Fanuc TP program (LS listing): CORR_NABI828_NIEO.LS

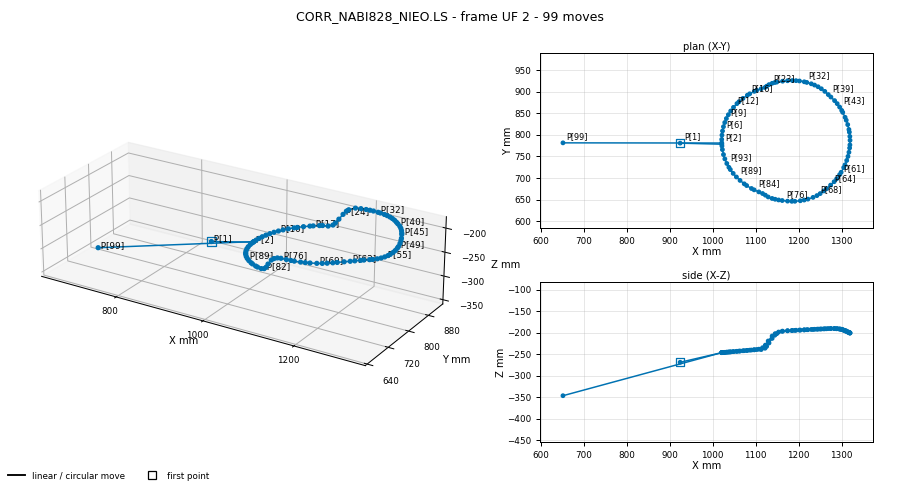
[picture p0: tool path of CORR_NABI828_NIEO.LS in frame UF 2, 99 of 99 moves have a stored position in this frame; points joined in program order, loops and branches not executed]
/PROG  CORR_NABI828_NIEO
/ATTR
OWNER		= MNEDITOR;
COMMENT		= "WeldPRO Auto-Gen";
PROG_SIZE	= 7125;
CREATE		= DATE 26-07-31  TIME 09:44:06;
MODIFIED	= DATE 26-07-31  TIME 10:09:20;
FILE_NAME	= CORR_NAB;
VERSION		= 0;
LINE_COUNT	= 113;
MEMORY_SIZE	= 7445;
PROTECT		= READ_WRITE;
TCD:  STACK_SIZE	= 0,
      TASK_PRIORITY	= 50,
      TIME_SLICE	= 0,
      BUSY_LAMP_OFF	= 0,
      ABORT_REQUEST	= 0,
      PAUSE_REQUEST	= 0;
DEFAULT_GROUP	= 1,*,*,*,*;
CONTROL_CODE	= 00000000 00000000;
/APPL
/MN
   1:  !WeldPRO Auto-Generated TPP ;
   2:  !TOR_XL_2026, TOR_xl_2907 ;
   3:   ;
   4:  UFRAME_NUM=2 ;
   5:  UTOOL_NUM=2 ;
   6:  !Feature Approach ;
   7:J P[1] 100% FINE    ;
   8:   ;
   9:  !Segment1 ;
  10:L P[2] 2000mm/sec FINE    ;
  11:   ;
  12:  CALL LASER_OFF    ;
  13:L P[3] R[23:moving]mm/sec CNT100    ;
  14:L P[4] R[23:moving]mm/sec CNT100    ;
  15:L P[5] R[23:moving]mm/sec CNT100    ;
  16:L P[6] R[23:moving]mm/sec CNT100    ;
  17:L P[7] R[23:moving]mm/sec CNT100    ;
  18:L P[8] R[23:moving]mm/sec CNT100    ;
  19:L P[9] R[23:moving]mm/sec CNT100    ;
  20:L P[10] R[23:moving]mm/sec CNT100    ;
  21:L P[11] R[23:moving]mm/sec CNT100    ;
  22:L P[12] R[23:moving]mm/sec CNT100    ;
  23:L P[13] R[23:moving]mm/sec CNT100    ;
  24:L P[14] R[23:moving]mm/sec CNT100    ;
  25:L P[15] R[23:moving]mm/sec CNT100    ;
  26:L P[16] R[23:moving]mm/sec CNT100    ;
  27:L P[17] R[23:moving]mm/sec CNT100    ;
  28:L P[18] R[23:moving]mm/sec CNT100    ;
  29:L P[19] R[23:moving]mm/sec CNT100    ;
  30:L P[20] R[23:moving]mm/sec CNT100    ;
  31:L P[21] R[23:moving]mm/sec CNT100    ;
  32:L P[22] R[23:moving]mm/sec CNT100    ;
  33:L P[23] R[23:moving]mm/sec CNT100    ;
  34:L P[24] R[23:moving]mm/sec CNT100    ;
  35:L P[25] R[23:moving]mm/sec CNT100    ;
  36:L P[26] R[23:moving]mm/sec CNT100    ;
  37:L P[27] R[23:moving]mm/sec CNT100    ;
  38:L P[28] R[23:moving]mm/sec CNT100    ;
  39:L P[29] R[23:moving]mm/sec CNT100    ;
  40:L P[30] R[23:moving]mm/sec CNT100    ;
  41:L P[31] R[23:moving]mm/sec CNT100    ;
  42:L P[32] R[23:moving]mm/sec CNT100    ;
  43:L P[33] R[23:moving]mm/sec CNT100    ;
  44:L P[34] R[23:moving]mm/sec CNT100    ;
  45:L P[35] R[23:moving]mm/sec CNT100    ;
  46:L P[36] R[23:moving]mm/sec CNT100    ;
  47:L P[37] R[23:moving]mm/sec CNT100    ;
  48:L P[38] R[23:moving]mm/sec CNT100    ;
  49:L P[39] R[23:moving]mm/sec CNT100    ;
  50:L P[40] R[23:moving]mm/sec CNT100    ;
  51:L P[41] R[23:moving]mm/sec CNT100    ;
  52:L P[42] R[23:moving]mm/sec CNT100    ;
  53:L P[43] R[23:moving]mm/sec CNT100    ;
  54:L P[44] R[23:moving]mm/sec CNT100    ;
  55:L P[45] R[23:moving]mm/sec CNT100    ;
  56:L P[46] R[23:moving]mm/sec CNT100    ;
  57:L P[47] R[23:moving]mm/sec CNT100    ;
  58:L P[48] R[23:moving]mm/sec CNT100    ;
  59:L P[49] R[23:moving]mm/sec CNT100    ;
  60:L P[50] R[23:moving]mm/sec CNT100    ;
  61:L P[51] R[23:moving]mm/sec CNT100    ;
  62:L P[52] R[23:moving]mm/sec CNT100    ;
  63:L P[53] R[23:moving]mm/sec CNT100    ;
  64:L P[54] R[23:moving]mm/sec CNT100    ;
  65:L P[55] R[23:moving]mm/sec CNT100    ;
  66:L P[56] R[23:moving]mm/sec CNT100    ;
  67:L P[57] R[23:moving]mm/sec CNT100    ;
  68:L P[58] R[23:moving]mm/sec CNT100    ;
  69:L P[59] R[23:moving]mm/sec CNT100    ;
  70:L P[60] R[23:moving]mm/sec CNT100    ;
  71:L P[61] R[23:moving]mm/sec CNT100    ;
  72:L P[62] R[23:moving]mm/sec CNT100    ;
  73:L P[63] R[23:moving]mm/sec CNT100    ;
  74:L P[64] R[23:moving]mm/sec CNT100    ;
  75:L P[65] R[23:moving]mm/sec CNT100    ;
  76:L P[66] R[23:moving]mm/sec CNT100    ;
  77:L P[67] R[23:moving]mm/sec CNT100    ;
  78:L P[68] R[23:moving]mm/sec CNT100    ;
  79:L P[69] R[23:moving]mm/sec CNT100    ;
  80:L P[70] R[23:moving]mm/sec CNT100    ;
  81:L P[71] R[23:moving]mm/sec CNT100    ;
  82:L P[72] R[23:moving]mm/sec CNT100    ;
  83:L P[73] R[23:moving]mm/sec CNT100    ;
  84:L P[74] R[23:moving]mm/sec CNT100    ;
  85:L P[75] R[23:moving]mm/sec CNT100    ;
  86:L P[76] R[23:moving]mm/sec CNT100    ;
  87:L P[77] R[23:moving]mm/sec CNT100    ;
  88:L P[78] R[23:moving]mm/sec CNT100    ;
  89:L P[79] R[23:moving]mm/sec CNT100    ;
  90:L P[80] R[23:moving]mm/sec CNT100    ;
  91:L P[81] R[23:moving]mm/sec CNT100    ;
  92:L P[82] R[23:moving]mm/sec CNT100    ;
  93:L P[83] R[23:moving]mm/sec CNT100    ;
  94:L P[84] R[23:moving]mm/sec CNT100    ;
  95:L P[85] R[23:moving]mm/sec CNT100    ;
  96:L P[86] R[23:moving]mm/sec CNT100    ;
  97:L P[87] R[23:moving]mm/sec CNT100    ;
  98:L P[88] R[23:moving]mm/sec CNT100    ;
  99:L P[89] R[23:moving]mm/sec CNT100    ;
 100:L P[90] R[23:moving]mm/sec CNT100    ;
 101:L P[91] R[23:moving]mm/sec CNT100    ;
 102:L P[92] R[23:moving]mm/sec CNT100    ;
 103:L P[93] R[23:moving]mm/sec CNT100    ;
 104:L P[94] R[23:moving]mm/sec CNT100    ;
 105:L P[95] R[23:moving]mm/sec CNT100    ;
 106:L P[96] R[23:moving]mm/sec CNT100    ;
 107:L P[97] R[23:moving]mm/sec CNT100    ;
 108:L P[98] R[23:moving]mm/sec FINE    ;
 109:  CALL LASER_OFF    ;
 110:   ;
 111:  !Feature Retreat ;
 112:L P[99] 2000mm/sec FINE    ;
 113:  CALL ROTATE    ;
/POS
P[1]{
   GP1:
	UF : 2, UT : 2,		CONFIG : 'F D T, 0, 0, 0',
	X =   924.335  mm,	Y =   780.986  mm,	Z =  -268.284  mm,
	W =  -106.495 deg,	P =   -15.000 deg,	R =    94.234 deg
};
P[2]{
   GP1:
	UF : 2, UT : 2,		CONFIG : 'F D T, 0, 0, 0',
	X =  1021.169  mm,	Y =   778.543  mm,	Z =  -245.849  mm,
	W =  -106.497 deg,	P =   -14.995 deg,	R =    94.216 deg
};
P[3]{
   GP1:
	UF : 2, UT : 2,		CONFIG : 'F D T, 0, 0, 0',
	X =  1021.011  mm,	Y =   781.278  mm,	Z =  -245.859  mm,
	W =  -106.499 deg,	P =   -14.997 deg,	R =    94.226 deg
};
P[4]{
   GP1:
	UF : 2, UT : 2,		CONFIG : 'F D T, 0, 0, 0',
	X =  1020.925  mm,	Y =   789.680  mm,	Z =  -245.860  mm,
	W =  -106.492 deg,	P =   -15.098 deg,	R =    90.372 deg
};
P[5]{
   GP1:
	UF : 2, UT : 2,		CONFIG : 'F D T, 0, 0, 0',
	X =  1021.526  mm,	Y =   799.646  mm,	Z =  -245.805  mm,
	W =  -106.481 deg,	P =   -15.218 deg,	R =    85.605 deg
};
P[6]{
   GP1:
	UF : 2, UT : 2,		CONFIG : 'F D T, 0, 0, 0',
	X =  1022.834  mm,	Y =   809.284  mm,	Z =  -245.689  mm,
	W =  -106.456 deg,	P =   -15.335 deg,	R =    80.815 deg
};
P[7]{
   GP1:
	UF : 2, UT : 2,		CONFIG : 'F D T, 0, 0, 0',
	X =  1025.009  mm,	Y =   819.272  mm,	Z =  -245.496  mm,
	W =  -106.423 deg,	P =   -15.450 deg,	R =    76.090 deg
};
P[8]{
   GP1:
	UF : 2, UT : 2,		CONFIG : 'F D T, 0, 0, 0',
	X =  1027.996  mm,	Y =   828.917  mm,	Z =  -245.233  mm,
	W =  -106.378 deg,	P =   -15.565 deg,	R =    71.217 deg
};
P[9]{
   GP1:
	UF : 2, UT : 2,		CONFIG : 'F D T, 0, 0, 0',
	X =  1031.797  mm,	Y =   838.208  mm,	Z =  -244.899  mm,
	W =  -106.322 deg,	P =   -15.679 deg,	R =    66.207 deg
};
P[10]{
   GP1:
	UF : 2, UT : 2,		CONFIG : 'F D T, 0, 0, 0',
	X =  1036.420  mm,	Y =   847.146  mm,	Z =  -244.496  mm,
	W =  -106.254 deg,	P =   -15.791 deg,	R =    61.015 deg
};
P[11]{
   GP1:
	UF : 2, UT : 2,		CONFIG : 'F D T, 0, 0, 0',
	X =  1041.832  mm,	Y =   855.675  mm,	Z =  -244.021  mm,
	W =  -106.177 deg,	P =   -15.894 deg,	R =    55.979 deg
};
P[12]{
   GP1:
	UF : 2, UT : 2,		CONFIG : 'F D T, 0, 0, 0',
	X =  1048.352  mm,	Y =   864.193  mm,	Z =  -243.446  mm,
	W =  -106.096 deg,	P =   -15.986 deg,	R =    51.162 deg
};
P[13]{
   GP1:
	UF : 2, UT : 2,		CONFIG : 'F D T, 0, 0, 0',
	X =  1056.339  mm,	Y =   872.875  mm,	Z =  -242.736  mm,
	W =  -106.012 deg,	P =   -16.066 deg,	R =    46.632 deg
};
P[14]{
   GP1:
	UF : 2, UT : 2,		CONFIG : 'F D T, 0, 0, 0',
	X =  1061.049  mm,	Y =   877.307  mm,	Z =  -242.336  mm,
	W =  -105.919 deg,	P =   -16.142 deg,	R =    41.952 deg
};
P[15]{
   GP1:
	UF : 2, UT : 2,		CONFIG : 'F D T, 0, 0, 0',
	X =  1070.354  mm,	Y =   885.100  mm,	Z =  -241.489  mm,
	W =  -105.870 deg,	P =   -16.177 deg,	R =    39.609 deg
};
P[16]{
   GP1:
	UF : 2, UT : 2,		CONFIG : 'F D T, 0, 0, 0',
	X =  1080.529  mm,	Y =   892.333  mm,	Z =  -240.579  mm,
	W =  -105.777 deg,	P =   -16.235 deg,	R =    35.365 deg
};
P[17]{
   GP1:
	UF : 2, UT : 2,		CONFIG : 'F D T, 0, 0, 0',
	X =  1086.008  mm,	Y =   895.696  mm,	Z =  -240.112  mm,
	W =  -105.677 deg,	P =   -16.289 deg,	R =    30.964 deg
};
P[18]{
   GP1:
	UF : 2, UT : 2,		CONFIG : 'F D T, 0, 0, 0',
	X =  1096.709  mm,	Y =   901.377  mm,	Z =  -239.157  mm,
	W =  -105.579 deg,	P =   -16.333 deg,	R =    26.830 deg
};
P[19]{
   GP1:
	UF : 2, UT : 2,		CONFIG : 'F D T, 0, 0, 0',
	X =  1102.228  mm,	Y =   903.878  mm,	Z =  -238.661  mm,
	W =  -105.536 deg,	P =   -16.344 deg,	R =    25.018 deg
};
P[20]{
   GP1:
	UF : 2, UT : 2,		CONFIG : 'F D T, 0, 0, 0',
	X =  1112.693  mm,	Y =   907.377  mm,	Z =  -238.660  mm,
	W =  -116.027 deg,	P =   -16.063 deg,	R =    30.267 deg
};
P[21]{
   GP1:
	UF : 2, UT : 2,		CONFIG : 'F D T, 0, 0, 0',
	X =  1121.614  mm,	Y =   910.523  mm,	Z =  -235.623  mm,
	W =  -126.877 deg,	P =   -15.356 deg,	R =    25.893 deg
};
P[22]{
   GP1:
	UF : 2, UT : 2,		CONFIG : 'F D T, 0, 0, 0',
	X =  1125.314  mm,	Y =   913.254  mm,	Z =  -231.338  mm,
	W =  -119.393 deg,	P =   -15.981 deg,	R =    16.221 deg
};
P[23]{
   GP1:
	UF : 2, UT : 2,		CONFIG : 'F D T, 0, 0, 0',
	X =  1130.886  mm,	Y =   916.988  mm,	Z =  -223.426  mm,
	W =  -115.329 deg,	P =   -16.208 deg,	R =    11.788 deg
};
P[24]{
   GP1:
	UF : 2, UT : 2,		CONFIG : 'F D T, 0, 0, 0',
	X =  1138.204  mm,	Y =   920.113  mm,	Z =  -212.785  mm,
	W =  -112.639 deg,	P =   -16.315 deg,	R =     9.714 deg
};
P[25]{
   GP1:
	UF : 2, UT : 2,		CONFIG : 'F D T, 0, 0, 0',
	X =  1144.373  mm,	Y =   921.944  mm,	Z =  -205.360  mm,
	W =  -110.015 deg,	P =   -16.386 deg,	R =     9.649 deg
};
P[26]{
   GP1:
	UF : 2, UT : 2,		CONFIG : 'F D T, 0, 0, 0',
	X =  1148.959  mm,	Y =   922.948  mm,	Z =  -201.734  mm,
	W =  -108.552 deg,	P =   -16.418 deg,	R =     8.950 deg
};
P[27]{
   GP1:
	UF : 2, UT : 2,		CONFIG : 'F D T, 0, 0, 0',
	X =  1162.494  mm,	Y =   925.003  mm,	Z =  -195.937  mm,
	W =  -105.409 deg,	P =   -16.443 deg,	R =     6.805 deg
};
P[28]{
   GP1:
	UF : 2, UT : 2,		CONFIG : 'F D T, 0, 0, 0',
	X =  1173.955  mm,	Y =   926.027  mm,	Z =  -194.869  mm,
	W =  -104.866 deg,	P =   -16.444 deg,	R =     5.597 deg
};
P[29]{
   GP1:
	UF : 2, UT : 2,		CONFIG : 'F D T, 0, 0, 0',
	X =  1185.153  mm,	Y =   926.452  mm,	Z =  -194.244  mm,
	W =  -104.887 deg,	P =   -16.444 deg,	R =     3.523 deg
};
P[30]{
   GP1:
	UF : 2, UT : 2,		CONFIG : 'F D T, 0, 0, 0',
	X =  1193.623  mm,	Y =   926.230  mm,	Z =  -193.803  mm,
	W =  -104.930 deg,	P =   -16.439 deg,	R =     -.729 deg
};
P[31]{
   GP1:
	UF : 2, UT : 2,		CONFIG : 'F D T, 0, 0, 0',
	X =  1201.657  mm,	Y =   925.491  mm,	Z =  -193.395  mm,
	W =  -104.979 deg,	P =   -16.424 deg,	R =    -5.541 deg
};
P[32]{
   GP1:
	UF : 2, UT : 2,		CONFIG : 'F D T, 0, 0, 0',
	X =  1212.836  mm,	Y =   923.579  mm,	Z =  -192.803  mm,
	W =  -105.028 deg,	P =   -16.400 deg,	R =   -10.259 deg
};
P[33]{
   GP1:
	UF : 2, UT : 2,		CONFIG : 'F D T, 0, 0, 0',
	X =  1218.699  mm,	Y =   922.145  mm,	Z =  -192.512  mm,
	W =  -105.070 deg,	P =   -16.371 deg,	R =   -14.490 deg
};
P[34]{
   GP1:
	UF : 2, UT : 2,		CONFIG : 'F D T, 0, 0, 0',
	X =  1229.137  mm,	Y =   918.943  mm,	Z =  -191.955  mm,
	W =  -105.112 deg,	P =   -16.334 deg,	R =   -18.515 deg
};
P[35]{
   GP1:
	UF : 2, UT : 2,		CONFIG : 'F D T, 0, 0, 0',
	X =  1236.713  mm,	Y =   916.001  mm,	Z =  -191.568  mm,
	W =  -105.158 deg,	P =   -16.285 deg,	R =   -23.051 deg
};
P[36]{
   GP1:
	UF : 2, UT : 2,		CONFIG : 'F D T, 0, 0, 0',
	X =  1244.878  mm,	Y =   912.086  mm,	Z =  -191.164  mm,
	W =  -105.219 deg,	P =   -16.204 deg,	R =   -29.417 deg
};
P[37]{
   GP1:
	UF : 2, UT : 2,		CONFIG : 'F D T, 0, 0, 0',
	X =  1252.474  mm,	Y =   907.445  mm,	Z =  -190.821  mm,
	W =  -105.311 deg,	P =   -16.047 deg,	R =   -39.415 deg
};
P[38]{
   GP1:
	UF : 2, UT : 2,		CONFIG : 'F D T, 0, 0, 0',
	X =  1260.559  mm,	Y =   901.318  mm,	Z =  -190.356  mm,
	W =  -105.307 deg,	P =   -16.055 deg,	R =   -38.974 deg
};
P[39]{
   GP1:
	UF : 2, UT : 2,		CONFIG : 'F D T, 0, 0, 0',
	X =  1268.657  mm,	Y =   893.885  mm,	Z =  -189.892  mm,
	W =  -105.302 deg,	P =   -16.063 deg,	R =   -38.625 deg
};
P[40]{
   GP1:
	UF : 2, UT : 2,		CONFIG : 'F D T, 0, 0, 0',
	X =  1274.729  mm,	Y =   888.161  mm,	Z =  -189.680  mm,
	W =  -105.469 deg,	P =   -15.944 deg,	R =   -44.976 deg
};
P[41]{
   GP1:
	UF : 2, UT : 2,		CONFIG : 'F D T, 0, 0, 0',
	X =  1283.312  mm,	Y =   879.865  mm,	Z =  -189.600  mm,
	W =  -105.661 deg,	P =   -15.890 deg,	R =   -47.714 deg
};
P[42]{
   GP1:
	UF : 2, UT : 2,		CONFIG : 'F D T, 0, 0, 0',
	X =  1289.348  mm,	Y =   872.830  mm,	Z =  -189.888  mm,
	W =  -106.210 deg,	P =   -15.792 deg,	R =   -52.259 deg
};
P[43]{
   GP1:
	UF : 2, UT : 2,		CONFIG : 'F D T, 0, 0, 0',
	X =  1294.988  mm,	Y =   864.946  mm,	Z =  -190.521  mm,
	W =  -106.927 deg,	P =   -15.688 deg,	R =   -56.663 deg
};
P[44]{
   GP1:
	UF : 2, UT : 2,		CONFIG : 'F D T, 0, 0, 0',
	X =  1299.851  mm,	Y =   857.005  mm,	Z =  -191.459  mm,
	W =  -107.603 deg,	P =   -15.597 deg,	R =   -60.243 deg
};
P[45]{
   GP1:
	UF : 2, UT : 2,		CONFIG : 'F D T, 0, 0, 0',
	X =  1302.244  mm,	Y =   852.538  mm,	Z =  -192.125  mm,
	W =  -108.271 deg,	P =   -15.504 deg,	R =   -63.685 deg
};
P[46]{
   GP1:
	UF : 2, UT : 2,		CONFIG : 'F D T, 0, 0, 0',
	X =  1307.708  mm,	Y =   841.061  mm,	Z =  -194.213  mm,
	W =  -109.144 deg,	P =   -15.377 deg,	R =   -68.203 deg
};
P[47]{
   GP1:
	UF : 2, UT : 2,		CONFIG : 'F D T, 0, 0, 0',
	X =  1310.369  mm,	Y =   834.284  mm,	Z =  -195.533  mm,
	W =  -109.899 deg,	P =   -15.253 deg,	R =   -72.505 deg
};
P[48]{
   GP1:
	UF : 2, UT : 2,		CONFIG : 'F D T, 0, 0, 0',
	X =  1313.804  mm,	Y =   824.052  mm,	Z =  -197.235  mm,
	W =  -110.273 deg,	P =   -15.181 deg,	R =   -74.981 deg
};
P[49]{
   GP1:
	UF : 2, UT : 2,		CONFIG : 'F D T, 0, 0, 0',
	X =  1316.610  mm,	Y =   812.754  mm,	Z =  -198.682  mm,
	W =  -110.635 deg,	P =   -14.305 deg,	R =   -78.232 deg
};
P[50]{
   GP1:
	UF : 2, UT : 2,		CONFIG : 'F D T, 0, 0, 0',
	X =  1317.639  mm,	Y =   806.573  mm,	Z =  -199.259  mm,
	W =  -111.054 deg,	P =   -14.769 deg,	R =   -83.164 deg
};
P[51]{
   GP1:
	UF : 2, UT : 2,		CONFIG : 'F D T, 0, 0, 0',
	X =  1318.762  mm,	Y =   796.603  mm,	Z =  -199.910  mm,
	W =  -111.190 deg,	P =   -15.305 deg,	R =   -88.308 deg
};
P[52]{
   GP1:
	UF : 2, UT : 2,		CONFIG : 'F D T, 0, 0, 0',
	X =  1319.192  mm,	Y =   787.630  mm,	Z =  -200.199  mm,
	W =  -111.129 deg,	P =   -15.645 deg,	R =   -91.614 deg
};
P[53]{
   GP1:
	UF : 2, UT : 2,		CONFIG : 'F D T, 0, 0, 0',
	X =  1318.902  mm,	Y =   776.906  mm,	Z =  -200.178  mm,
	W =  -110.757 deg,	P =   -14.624 deg,	R =   -96.575 deg
};
P[54]{
   GP1:
	UF : 2, UT : 2,		CONFIG : 'F D T, 0, 0, 0',
	X =  1318.207  mm,	Y =   769.725  mm,	Z =  -199.914  mm,
	W =  -110.276 deg,	P =   -14.535 deg,	R =  -100.836 deg
};
P[55]{
   GP1:
	UF : 2, UT : 2,		CONFIG : 'F D T, 0, 0, 0',
	X =  1316.644  mm,	Y =   759.802  mm,	Z =  -199.267  mm,
	W =  -109.635 deg,	P =   -14.447 deg,	R =  -105.265 deg
};
P[56]{
   GP1:
	UF : 2, UT : 2,		CONFIG : 'F D T, 0, 0, 0',
	X =  1314.412  mm,	Y =   750.198  mm,	Z =  -198.320  mm,
	W =  -109.083 deg,	P =   -14.382 deg,	R =  -108.625 deg
};
P[57]{
   GP1:
	UF : 2, UT : 2,		CONFIG : 'F D T, 0, 0, 0',
	X =  1311.482  mm,	Y =   740.798  mm,	Z =  -197.069  mm,
	W =  -108.349 deg,	P =   -14.302 deg,	R =  -112.873 deg
};
P[58]{
   GP1:
	UF : 2, UT : 2,		CONFIG : 'F D T, 0, 0, 0',
	X =  1307.481  mm,	Y =   730.593  mm,	Z =  -195.358  mm,
	W =  -107.748 deg,	P =   -14.239 deg,	R =  -116.265 deg
};
P[59]{
   GP1:
	UF : 2, UT : 2,		CONFIG : 'F D T, 0, 0, 0',
	X =  1304.470  mm,	Y =   724.222  mm,	Z =  -194.103  mm,
	W =  -106.924 deg,	P =   -14.148 deg,	R =  -121.191 deg
};
P[60]{
   GP1:
	UF : 2, UT : 2,		CONFIG : 'F D T, 0, 0, 0',
	X =  1298.511  mm,	Y =   713.296  mm,	Z =  -192.122  mm,
	W =  -106.269 deg,	P =   -14.066 deg,	R =  -125.698 deg
};
P[61]{
   GP1:
	UF : 2, UT : 2,		CONFIG : 'F D T, 0, 0, 0',
	X =  1294.971  mm,	Y =   707.729  mm,	Z =  -191.348  mm,
	W =  -105.781 deg,	P =   -13.988 deg,	R =  -130.143 deg
};
P[62]{
   GP1:
	UF : 2, UT : 2,		CONFIG : 'F D T, 0, 0, 0',
	X =  1288.025  mm,	Y =   698.069  mm,	Z =  -190.397  mm,
	W =  -105.527 deg,	P =   -13.913 deg,	R =  -134.519 deg
};
P[63]{
   GP1:
	UF : 2, UT : 2,		CONFIG : 'F D T, 0, 0, 0',
	X =  1282.229  mm,	Y =   691.364  mm,	Z =  -190.048  mm,
	W =  -105.437 deg,	P =   -13.849 deg,	R =  -138.629 deg
};
P[64]{
   GP1:
	UF : 2, UT : 2,		CONFIG : 'F D T, 0, 0, 0',
	X =  1274.067  mm,	Y =   683.450  mm,	Z =  -189.989  mm,
	W =  -105.429 deg,	P =   -13.831 deg,	R =  -139.837 deg
};
P[65]{
   GP1:
	UF : 2, UT : 2,		CONFIG : 'F D T, 0, 0, 0',
	X =  1264.393  mm,	Y =   675.114  mm,	Z =  -190.372  mm,
	W =  -105.443 deg,	P =   -13.863 deg,	R =  -137.727 deg
};
P[66]{
   GP1:
	UF : 2, UT : 2,		CONFIG : 'F D T, 0, 0, 0',
	X =  1258.094  mm,	Y =   669.886  mm,	Z =  -190.658  mm,
	W =  -105.373 deg,	P =   -13.729 deg,	R =  -147.436 deg
};
P[67]{
   GP1:
	UF : 2, UT : 2,		CONFIG : 'F D T, 0, 0, 0',
	X =  1249.807  mm,	Y =   663.762  mm,	Z =  -191.053  mm,
	W =  -105.298 deg,	P =   -13.637 deg,	R =  -156.529 deg
};
P[68]{
   GP1:
	UF : 2, UT : 2,		CONFIG : 'F D T, 0, 0, 0',
	X =  1242.212  mm,	Y =   659.104  mm,	Z =  -191.465  mm,
	W =  -105.277 deg,	P =   -13.618 deg,	R =  -158.976 deg
};
P[69]{
   GP1:
	UF : 2, UT : 2,		CONFIG : 'F D T, 0, 0, 0',
	X =  1233.218  mm,	Y =   654.986  mm,	Z =  -191.945  mm,
	W =  -105.241 deg,	P =   -13.592 deg,	R =  -162.969 deg
};
P[70]{
   GP1:
	UF : 2, UT : 2,		CONFIG : 'F D T, 0, 0, 0',
	X =  1221.263  mm,	Y =   650.913  mm,	Z =  -192.596  mm,
	W =  -105.203 deg,	P =   -13.573 deg,	R =  -167.022 deg
};
P[71]{
   GP1:
	UF : 2, UT : 2,		CONFIG : 'F D T, 0, 0, 0',
	X =  1212.602  mm,	Y =   648.759  mm,	Z =  -193.048  mm,
	W =  -105.159 deg,	P =   -13.560 deg,	R =  -171.569 deg
};
P[72]{
   GP1:
	UF : 2, UT : 2,		CONFIG : 'F D T, 0, 0, 0',
	X =  1203.599  mm,	Y =   647.135  mm,	Z =  -193.518  mm,
	W =  -105.113 deg,	P =   -13.556 deg,	R =  -176.312 deg
};
P[73]{
   GP1:
	UF : 2, UT : 2,		CONFIG : 'F D T, 0, 0, 0',
	X =  1191.013  mm,	Y =   645.918  mm,	Z =  -194.198  mm,
	W =  -105.068 deg,	P =   -13.561 deg,	R =   179.213 deg
};
P[74]{
   GP1:
	UF : 2, UT : 2,		CONFIG : 'F D T, 0, 0, 0',
	X =  1183.845  mm,	Y =   645.822  mm,	Z =  -194.579  mm,
	W =  -105.038 deg,	P =   -13.569 deg,	R =   176.231 deg
};
P[75]{
   GP1:
	UF : 2, UT : 2,		CONFIG : 'F D T, 0, 0, 0',
	X =  1173.939  mm,	Y =   646.265  mm,	Z =  -195.168  mm,
	W =  -105.207 deg,	P =   -13.572 deg,	R =   175.290 deg
};
P[76]{
   GP1:
	UF : 2, UT : 2,		CONFIG : 'F D T, 0, 0, 0',
	X =  1161.575  mm,	Y =   647.632  mm,	Z =  -196.165  mm,
	W =  -107.012 deg,	P =   -13.569 deg,	R =   174.537 deg
};
P[77]{
   GP1:
	UF : 2, UT : 2,		CONFIG : 'F D T, 0, 0, 0',
	X =  1153.168  mm,	Y =   648.973  mm,	Z =  -197.975  mm,
	W =  -109.414 deg,	P =   -13.538 deg,	R =   174.483 deg
};
P[78]{
   GP1:
	UF : 2, UT : 2,		CONFIG : 'F D T, 0, 0, 0',
	X =  1145.177  mm,	Y =   650.610  mm,	Z =  -201.789  mm,
	W =  -112.196 deg,	P =   -13.466 deg,	R =   175.323 deg
};
P[79]{
   GP1:
	UF : 2, UT : 2,		CONFIG : 'F D T, 0, 0, 0',
	X =  1138.128  mm,	Y =   652.473  mm,	Z =  -207.272  mm,
	W =  -114.872 deg,	P =   -13.369 deg,	R =   175.422 deg
};
P[80]{
   GP1:
	UF : 2, UT : 2,		CONFIG : 'F D T, 0, 0, 0',
	X =  1128.978  mm,	Y =   655.939  mm,	Z =  -218.803  mm,
	W =  -120.114 deg,	P =   -13.109 deg,	R =   172.293 deg
};
P[81]{
   GP1:
	UF : 2, UT : 2,		CONFIG : 'F D T, 0, 0, 0',
	X =  1122.387  mm,	Y =   660.121  mm,	Z =  -228.369  mm,
	W =  -126.809 deg,	P =   -12.620 deg,	R =   167.792 deg
};
P[82]{
   GP1:
	UF : 2, UT : 2,		CONFIG : 'F D T, 0, 0, 0',
	X =  1115.888  mm,	Y =   663.919  mm,	Z =  -234.412  mm,
	W =  -119.561 deg,	P =   -13.285 deg,	R =   157.806 deg
};
P[83]{
   GP1:
	UF : 2, UT : 2,		CONFIG : 'F D T, 0, 0, 0',
	X =  1107.226  mm,	Y =   667.706  mm,	Z =  -237.847  mm,
	W =  -107.219 deg,	P =   -13.741 deg,	R =   154.408 deg
};
P[84]{
   GP1:
	UF : 2, UT : 2,		CONFIG : 'F D T, 0, 0, 0',
	X =  1096.247  mm,	Y =   672.464  mm,	Z =  -239.251  mm,
	W =  -105.746 deg,	P =   -13.749 deg,	R =   154.142 deg
};
P[85]{
   GP1:
	UF : 2, UT : 2,		CONFIG : 'F D T, 0, 0, 0',
	X =  1090.096  mm,	Y =   675.636  mm,	Z =  -239.807  mm,
	W =  -105.804 deg,	P =   -13.784 deg,	R =   151.506 deg
};
P[86]{
   GP1:
	UF : 2, UT : 2,		CONFIG : 'F D T, 0, 0, 0',
	X =  1078.886  mm,	Y =   682.462  mm,	Z =  -240.821  mm,
	W =  -105.885 deg,	P =   -13.838 deg,	R =   147.739 deg
};
P[87]{
   GP1:
	UF : 2, UT : 2,		CONFIG : 'F D T, 0, 0, 0',
	X =  1073.285  mm,	Y =   686.490  mm,	Z =  -241.298  mm,
	W =  -105.988 deg,	P =   -13.918 deg,	R =   142.681 deg
};
P[88]{
   GP1:
	UF : 2, UT : 2,		CONFIG : 'F D T, 0, 0, 0',
	X =  1063.552  mm,	Y =   694.409  mm,	Z =  -242.147  mm,
	W =  -106.084 deg,	P =   -14.001 deg,	R =   137.677 deg
};
P[89]{
   GP1:
	UF : 2, UT : 2,		CONFIG : 'F D T, 0, 0, 0',
	X =  1055.102  mm,	Y =   702.364  mm,	Z =  -242.855  mm,
	W =  -106.129 deg,	P =   -14.056 deg,	R =   135.015 deg
};
P[90]{
   GP1:
	UF : 2, UT : 2,		CONFIG : 'F D T, 0, 0, 0',
	X =  1047.622  mm,	Y =   710.709  mm,	Z =  -243.534  mm,
	W =  -106.186 deg,	P =   -14.117 deg,	R =   131.622 deg
};
P[91]{
   GP1:
	UF : 2, UT : 2,		CONFIG : 'F D T, 0, 0, 0',
	X =  1040.978  mm,	Y =   719.601  mm,	Z =  -244.130  mm,
	W =  -106.269 deg,	P =   -14.239 deg,	R =   125.999 deg
};
P[92]{
   GP1:
	UF : 2, UT : 2,		CONFIG : 'F D T, 0, 0, 0',
	X =  1037.623  mm,	Y =   724.905  mm,	Z =  -244.406  mm,
	W =  -106.343 deg,	P =   -14.367 deg,	R =   120.225 deg
};
P[93]{
   GP1:
	UF : 2, UT : 2,		CONFIG : 'F D T, 0, 0, 0',
	X =  1032.783  mm,	Y =   733.762  mm,	Z =  -244.809  mm,
	W =  -106.383 deg,	P =   -14.448 deg,	R =   116.672 deg
};
P[94]{
   GP1:
	UF : 2, UT : 2,		CONFIG : 'F D T, 0, 0, 0',
	X =  1028.249  mm,	Y =   744.359  mm,	Z =  -245.192  mm,
	W =  -106.433 deg,	P =   -14.556 deg,	R =   111.957 deg
};
P[95]{
   GP1:
	UF : 2, UT : 2,		CONFIG : 'F D T, 0, 0, 0',
	X =  1025.060  mm,	Y =   754.472  mm,	Z =  -245.491  mm,
	W =  -106.465 deg,	P =   -14.714 deg,	R =   105.666 deg
};
P[96]{
   GP1:
	UF : 2, UT : 2,		CONFIG : 'F D T, 0, 1, 0',
	X =  1022.562  mm,	Y =   766.062  mm,	Z =  -245.746  mm,
	W =  -106.480 deg,	P =   -14.798 deg,	R =   102.261 deg
};
P[97]{
   GP1:
	UF : 2, UT : 2,		CONFIG : 'F D T, 0, 1, 0',
	X =  1021.496  mm,	Y =   774.371  mm,	Z =  -245.829  mm,
	W =  -106.494 deg,	P =   -14.935 deg,	R =    96.827 deg
};
P[98]{
   GP1:
	UF : 2, UT : 2,		CONFIG : 'F D T, 0, 1, 0',
	X =  1021.011  mm,	Y =   781.277  mm,	Z =  -245.859  mm,
	W =  -106.501 deg,	P =   -15.000 deg,	R =    94.236 deg
};
P[99]{
   GP1:
	UF : 2, UT : 2,		CONFIG : 'F D T, 0, 1, 0',
	X =   651.995  mm,	Y =   781.694  mm,	Z =  -345.952  mm,
	W =  -106.495 deg,	P =   -15.000 deg,	R =    94.234 deg
};
/END
